(* IEC 61131-3 sources: repolevel_ST_code_completion/output/0122完整版本_无planner目前sota/repoeval_four-level_elevator_control/readful_result_no_provide, 3 files *)

(* ---- F_CheckJobInDirection.st ---- *)
VAR
	i	:	USINT;
END_VAR

F_CheckJobInDirection := FALSE;

IF bIncreasing THEN
	// 向上检查（从低楼层到高楼层）
	FOR i := nStartFloor TO nEndFloor DO
		IF Tar_Dir.IsStopFloor[i] THEN
			F_CheckJobInDirection := TRUE;
			RETURN;
		END_IF
	END_FOR
ELSE
	// 向下检查（从高楼层到低楼层）
	FOR i := nEndFloor TO nStartFloor BY -1 DO
		IF Tar_Dir.IsStopFloor[i] THEN
			F_CheckJobInDirection := TRUE;
			RETURN;
		END_IF
	END_FOR
END_IF;

RETURN;
END_FUNCTION

(* ---- F_ClearFloorStop.st ---- *)
VAR
	MaxNumFloor : USINT := 4; // Maximum number of floors
END_VAR

// Clear upward stop indicator
IF bClearUpStop AND (nFloor >= 1 AND nFloor <= MaxNumFloor - 1) THEN
  Tar_Dir.IsUpStop[nFloor] := FALSE;
  QFloorUpLed[nFloor] := FALSE;
END_IF

// Clear downward stop indicator
IF bClearDownStop AND (nFloor >= 2 AND nFloor <= MaxNumFloor) THEN
  Tar_Dir.IsDownStop[nFloor] := FALSE;
  QFloorDownLed[nFloor] := FALSE;
END_IF

// Clear floor stop indicator
IF bClearStopFloor AND (nFloor >= 1 AND nFloor <= MaxNumFloor) THEN
  Tar_Dir.IsStopFloor[nFloor] := FALSE;
  QGoFloorLed[nFloor] := FALSE;
END_IF

RETURN;
END_FUNCTION

(* ---- F_SetElevatorDirection.st ---- *)
VAR
	bDirectionSet	:	BOOL;		//方向是否已设置
END_VAR

bDirectionSet := FALSE;

IF nTargetFloor > nCurrentFloor THEN
	// 目标楼层高于当前楼层，电梯上升
	Tar_Dir.IsPositive := TRUE;
	Tar_Dir.IsNegative := FALSE;
	bDirectionSet := TRUE;
ELSIF nTargetFloor < nCurrentFloor THEN
	// 目标楼层低于当前楼层，电梯下降
	Tar_Dir.IsPositive := FALSE;
	Tar_Dir.IsNegative := TRUE;
	bDirectionSet := TRUE;
END_IF

RETURN;
END_FUNCTION
